INTERFACE I_SnappyVerify

PROPERTY stVerificationResult : REFERENCE TO ST_VerificationResult
GET
END_GET
END_PROPERTY

METHOD Verify : HRESULT
VAR_INPUT
	anyArg	: ANY;
END_VAR
END_METHOD

END_INTERFACE

(* stored: Version 1.1.0.1, ProductVersion 3.1.4026.18
   Itf I_SnappyVerify: Id {7c2c6182-0b25-4b12-8e3e-a5d4788a1cc2}
   Property stVerificationResult: Id {821698e1-b21e-4444-ae08-c86776e1021b}
   Get Get: Id {6a2c1ceb-be10-47f7-b7b9-9b9684158924}
   Method Verify: Id {609ab44f-90dd-4019-a39e-31ae681b76a2} *)
